(* CODESYS project Uppgift 7.project

Project tree, tasks and I/O mapping:
  Device : CODESYS Control Win V3, 3S - Smart Software Solutions GmbH, order no. 305021, version 3.5.10.40
    application Application
      libraries: Standard, * (System)
      task MainTask (cyclic, interval t#20ms, priority 1) calls PLC_PRG
      task VISU_TASK (cyclic, interval 100 ms, priority 31) calls VisuElems.Visu_Prg
      program PLC_PRG [LD]
      visualisation Visualization
      global variables GVL
  libraries: VisuSymbols, 3.5.10.0 (System)
  text list GlobalTextList
*)

// Device/Application/GVL
{attribute 'qualified_only'}
VAR_GLOBAL
	Lamp_Green: BOOL;
	Lamp_Blue: BOOL;
	Btn_1: BOOL;
	TON_0: TON;
	TimerElisped_time: TIME;
	TimerElisped_time_2: TIME;
	TOF_0: TOF;
END_VAR

// Device/Application/PLC_PRG
PROGRAM PLC_PRG
VAR
	
END_VAR

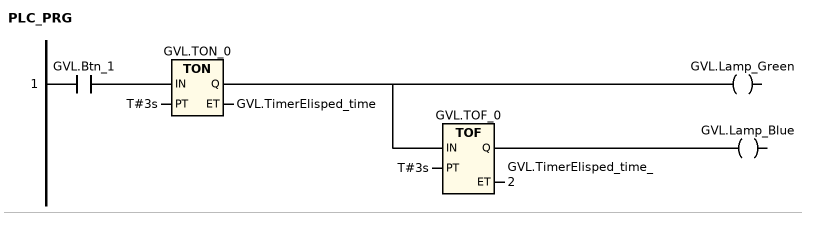
// NETWORK 1
GVL.TON_0(IN := GVL.Btn_1, PT := T#3s, ET => GVL.TimerElisped_time); // TON
GVL.Lamp_Green := GVL.TON_0.Q;
GVL.TOF_0(IN := GVL.TON_0.Q, PT := T#3s, ET => GVL.TimerElisped_time_2); // TOF
GVL.Lamp_Blue := GVL.TOF_0.Q;

END_PROGRAM

// Device/Application/Visualization
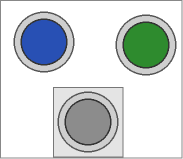
VISUALIZATION Visualization  // 183x159
    Lamp1 (9,7 70x70), variable: GVL.Lamp_Blue, style: Lamp-Lamp1-Blue
    Lamp1 (111,10 70x70), variable: GVL.Lamp_Green, style: Lamp-Lamp1-Green
    PushSwitch (53,87 70x70), variable: GVL.Btn_1, behaviour: TOGGLE, style: Switch-PushSwitch-Gray
END_VISUALIZATION
